// TIA Portal V18 program export: 2 tag tables, 0 data types, 0 data blocks, 1 code blocks (in call order from the OBs), 0 instance data blocks

VAR_GLOBAL   // PLC tag table "INGRESSI"
   In_1 AT %I1.0 : Bool;
   In_2 AT %I1.1 : Bool;
   In_3 AT %I1.2 : Bool;
   In_4 AT %I1.3 : Bool;
   In_5 AT %I1.4 : Bool;
   In_6 AT %I1.5 : Bool;
   In AT %IB1 : Byte;
END_VAR

VAR_GLOBAL   // PLC tag table "USCITE"
   Out_1 AT %Q0.0 : Bool;
   Out_2 AT %Q0.1 : Bool;
   Out_3 AT %Q0.2 : Bool;
   Out_4 AT %Q0.3 : Bool;
   Out_5 AT %Q0.4 : Bool;
   Var AT %Q0.5 : Bool;
END_VAR

ORGANIZATION_BLOCK "Main"   // OB1, LAD, ProgramCycle
TITLE = "Main Program Sweep (Cycle)"
{ S7_Optimized_Access := 'TRUE' }
// stored: SetENOAutomatically false
   VAR_INPUT
      Initial_Call : Bool;   // Initial call of this OB
      Remanence : Bool;   // =True, if remanent data are available
   END_VAR
BEGIN
END_ORGANIZATION_BLOCK
